Fanuc KAREL source: kb00192.KL

-- PROVISIONAL review KL for V770-1; original PC SHA256 a36524d791c438f337e23217461f13a3f51bcc81d2934dcd43d3d9906936395b
-- Incomplete behavior may be omitted. Consult companion uncertainty JSON. Do not deploy.
PROGRAM KB00192
%NOLOCKGROUP
VAR
  P1 : REAL
  RESULT : INTEGER
BEGIN
  -- UNRESOLVED_PC offsets 5-16; opcodes 2E,23
  -- UNRESOLVED_PC offsets 21-36; opcodes 27,22,76,23
  -- UNRESOLVED_PC offsets 41-45; opcodes 7F
END KB00192
